Universal Robots PolyScope program: barreraVirtualEsferaPROVAsetTCP.urp

Program barreraVirtualEsferaPROVAsetTCP (installation=defaultEsferaTCPs directory=/home/ur/ursim-current/programs/provesTFGmireia/new folder createdIn=5.15.1 lastSavedIn=5.15.1 robotSerialNumber=20195399999)
Calibrated DH parameters: a=[0, -0.24355, -0.2132, 0, 0, 0]; d=[0.15185, 0, 0, 0.13105, 0.08535, 0.0921]; alpha=[1.570796, 0, 0, 1.570796, -1.570796, 0]; deltaTheta=[0, 0, 0, 0, 0, 0]
InitVariablesNode
Robot Program (runOnlyOnce=true)
  'Definim dues surtTcp i surtToolFlange com a False per indicar quan es passa el limit.'
  surtTcp := False
  surtToolFlange := False
  surtMig := False
  'Indiquem les coordenades del centre de l'esfera.'
  centre := p[-0.017,-0.392,0.236,0,0,0]
  'Indiquem la variable de radi que te l'esfera.'
  radi := 0.3
  'Donem valor als radis del TCP,del punt del flange de l'eina i el punt mig.'
  radiTCP := 0.05
  radiMig := 0.09
  radiFlange := 0.06
  'Activem el moviment lliure.'
  Script: freedrive_mode()
  Loop Forever
    If surtTcp≟ True  or (surtTcp≟ True  and surtToolFlange≟ True ) (checkContinuously=true)
      'La condicio es compleix, estem intentant superar la barrera virtual amb el TCP o tant amb el TCP com el flange.'
      'Aturem el moviment lliure.'
      Script: end_freedrive_mode()
      'Obtenim la posició del TCP per quedar-nos amb els graus dels joints.'
      Set DigitalOutput tcp=TCP_Eina; pin=digital_out[0]; digitalValue=1
      SetPayload (workpieceName=Payload_TCPEina payloadTransitionTime=0)
      puntAct := get_actual_tcp_pose()
      'Cridem el subprograma que rectifica la posicio de l'eina.'
      Call rectificarPosicio
      'Ara ja tornem a estar a dins l'area de moviment permesa, surtTCP li donem False.'
      surtTcp := False
      'Estem dins la condició que també poden estar tocant els dos, per tant, posem a fals surtToolFlange també.'
      surtToolFlange := False
    If surtToolFlange≟ True (checkContinuously=true)
      'La condicio es compleix, estem intentant superar la barrera virtual amb el cap de l'eina. '
      'Aturem el moviment lliure.'
      Script: end_freedrive_mode()
      'Obtenim la posició del flange de l'eina per quedar-nos amb els graus dels joints.'
      Set DigitalOutput tcp=CapEina; pin=digital_out[0]; digitalValue=1
      SetPayload (workpieceName=Payload_CapEina payloadTransitionTime=0)
      puntAct := get_actual_tcp_pose()
      'Cridem el subprograma que rectifica la posicio de l'eina.'
      Call rectificarPosicio
      'Ara ja tornem a estar a dins l'area de moviment permesa, surtToolFlange li donem False.'
      surtToolFlange := False
    If surtMig≟ True (checkContinuously=true)
      'La condicio es compleix, estem intentant superar la barrera virtual amb el punt del mig de l'eina. '
      'Aturem el moviment lliure.'
      Script: end_freedrive_mode()
      'Obtenim la posició del punt del mig de l'eina.'
      Set DigitalOutput tcp=TCP_Eina; pin=digital_out[0]; digitalValue=1
      SetPayload (workpieceName=Payload_TCPEina payloadTransitionTime=0)
      tcpActual := get_actual_tcp_pose()
      Set DigitalOutput tcp=CapEina; pin=digital_out[0]; digitalValue=1
      SetPayload (workpieceName=Payload_CapEina payloadTransitionTime=0)
      toolFlangeAct := get_actual_tcp_pose()
      puntAct := p[(tcpActual[0]+toolFlangeAct[0])/2,(tcpActual[1]+toolFlangeAct[1])/2,(tcpActual[2]+toolFlangeAct[2])/2,tcpActual[3],tcpActual[4],tcpActual[5]]
      'Cridem el subprograma que rectifica la posicio de l'eina.'
      Call rectificarPosicio
      'Ara ja tornem a estar a dins l'area de moviment permesa, surtMig li donem False.'
      surtMig := False
    Wait Sleep waitTime=0.01
SubProgram -> rectificarPosicio
Thread Thread_1 (runOnlyOnce=false)
  Loop Forever
    'Obtenim les posicions del TCP i el cap de l'eina.'
    Set DigitalOutput tcp=TCP_Eina; pin=digital_out[0]; digitalValue=1
    SetPayload (workpieceName=Payload_TCPEina payloadTransitionTime=0)
    llistaPosTCP := get_actual_tcp_pose()
    Set DigitalOutput tcp=CapEina; pin=digital_out[0]; digitalValue=1
    SetPayload (workpieceName=Payload_CapEina payloadTransitionTime=0)
    llistaPosTool := get_actual_tcp_pose()
    'Obtenim el punt intermig.'
    llistaPosMig := p[(llistaPosTCP[0]+llistaPosTool[0])/2,(llistaPosTCP[1]+llistaPosTool[1])/2,(llistaPosTCP[2]+llistaPosTool[2])/2,llistaPosTCP[3],llistaPosTCP[4],llistaPosTCP[5]]
    'Calculem la distancia entre dos punts, el centre i el tcp, toolFlange o punt del mig.'
    distPunts := radiTCP+sqrt(pow(llistaPosTCP[0]-centre[0],2)+pow(llistaPosTCP[1]-centre[1],2)+pow(llistaPosTCP[2]-centre[2],2))
    distPuntTool := radiFlange+ sqrt(pow(llistaPosTool[0]-centre[0],2)+pow(llistaPosTool[1]-centre[1],2)+pow(llistaPosTool[2]-centre[2],2))
    distPuntMig := radiMig+sqrt(pow(llistaPosMig[0]-centre[0],2)+pow(llistaPosMig[1]-centre[1],2)+pow(llistaPosMig[2]-centre[2],2))
    'Si la distancia calculada supera el valor radi, entrem a la condicio perque estem intentant superar el limit.'
    If distPunts≥radi or distPunts≤-radi (checkContinuously=true)
      'Supera el límit amb el TCP'
      surtTcp := True
    If distPuntTool≥radi or distPuntTool≤-radi (checkContinuously=true)
      'Supera el límit amb el flange de l'eina.'
      surtToolFlange := True
    If distPuntMig≥radi or distPuntMig≤-radi (checkContinuously=true)
      'Supera el límit amb el punt mig.'
      surtMig := True
    'Dins un loop que pot estar sense fer res varies vegades, sempres es millor indicar-li un wait.'
    Wait Sleep waitTime=0.01
SubProgram rectificarPosicio (keepSynchronizedWithDisk=false)
  'Subprograma cridat per tal de realitzar un moviment en una direccio concreta.'
  'Abans de ser cridat, cal haver obtingut la la posicio actual d'interès per tal de fer el moviment.'
  'Generem el vector director per anar des del punt actual de l'eina fins al centre.'
  vectorDir := [centre[0]-puntAct[0],centre[1]-puntAct[1],centre[2]-puntAct[2]]
  'Apliquem un Wait per tal de deixar temps per pensar,sino es mou alla on li vagi.'
  Wait Sleep waitTime=0.01
  'Ens movem en direcció el centre fins que s'hagi recorregut uns determinats mm.'
  MoveL speed 25 mm/s, acceleration 150 mm/s^2 (useActiveTCP=true) feature=Base
    MoveDirectionNode expression=vectorDir
      Until DISTANCE (allowActions=false deceleration=3 distanceNodeType=STOP) Distance=0.001; motionParameters(blendRadius=0)
  'Tornem a activar el moviment.'
  Script: freedrive_mode()
